INTERFACE I_StringBuilder

METHOD Append : I_StringBuilder
VAR_INPUT
	Value : T_MaxString;
END_VAR
END_METHOD

METHOD AppendAny : I_StringBuilder
VAR_INPUT
	Value : ANY;
END_VAR
END_METHOD

PROPERTY BufferAddress : POINTER TO BYTE
GET
END_GET
END_PROPERTY

METHOD Clear : I_StringBuilder
VAR_INPUT
END_VAR
END_METHOD

END_INTERFACE

(* stored: Version 1.1.0.1, ProductVersion 3.1.4024.13
   Itf I_StringBuilder: Id {01f8af8d-11f8-07a0-05e0-25e4eaaffbdc}
   Method Append: Id {60983611-7ee1-476d-88da-748e90a67f65}
   Method AppendAny: Id {72ed47cb-a9b5-4750-8215-27eb388814e0}
   Property BufferAddress: Id {64b43a8a-a0cd-44c9-86f9-68fa3df3b829}
   Get Get: Id {eaea8831-93e0-4747-86f9-01027dc93c3b}
   Method Clear: Id {5bd9befe-3ca8-4ef3-a795-849de7551fbf} *)
